{attribute 'linkalways'} 
{attribute 'no_explicit_call' := 'This FB is a CLASS and must be accessed using methods or properties'}
{attribute 'enable_dynamic_creation'}
FUNCTION_BLOCK _ETcVnContourApproximationMethod EXTENDS EnumDatatypeBase
VAR
	localData : ETcVnContourApproximationMethod;
	activeData : REFERENCE TO ETcVnContourApproximationMethod;
	enumBaseDatatype : _DINT(localData);
END_VAR

METHOD PRIVATE AddLocalEnumeration
VAR_INPUT
	Enumeration : T_MAXSTRING;
	Value : ETcVnContourApproximationMethod;
END_VAR
AddEnumeration(Enumeration, Value);
END_METHOD

PROPERTY PUBLIC Address : PVOID
GET
Address := ADR(activeData);
END_GET
END_PROPERTY

METHOD PUBLIC ClearReference
VAR_INPUT
END_VAR
activeData REF= localData;
SetBaseDatatypeReference();
END_METHOD

METHOD PUBLIC Clone : I_Datatype
VAR
    pClone : POINTER TO _ETcVnContourApproximationMethod;
END_VAR
pClone := __NEW(_ETcVnContourApproximationMethod(InitialValue := Value));
Clone := pClone^;
END_METHOD

METHOD FB_init : BOOL
VAR_INPUT
	bInitRetains : BOOL; // if TRUE, the retain variables are initialized (warm start / cold start)
	bInCopyCode : BOOL;  // if TRUE, the instance afterwards gets moved into the copy code (online change)
	InitialValue : ETcVnContourApproximationMethod;
END_VAR
localData := InitialValue;
AddBaseDatatype(enumBaseDatatype);
ClearReference();

AddLocalEnumeration('TCVN_CAM_NONE', ETcVnContourApproximationMethod.TCVN_CAM_NONE);
AddLocalEnumeration('TCVN_CAM_SIMPLE', ETcVnContourApproximationMethod.TCVN_CAM_SIMPLE);
AddLocalEnumeration('TCVN_CAM_TC89_L1', ETcVnContourApproximationMethod.TCVN_CAM_TC89_L1);
AddLocalEnumeration('TCVN_CAM_TC89_KCOS', ETcVnContourApproximationMethod.TCVN_CAM_TC89_KCOS);
END_METHOD

PROPERTY PUBLIC Identifier : T_MAXSTRING
GET
Identifier := 'ETcVnContourApproximationMethod';
END_GET
END_PROPERTY

METHOD IsEnumeratorValueEqual : BOOL
VAR_INPUT
	Enumerator : I_KeyValueForwardEnumerator;
END_VAR
VAR
	storedValue : ETcVnContourApproximationMethod;
END_VAR
IF NOT Enumerator.TryGet(storedValue) THEN
	RETURN;
END_IF

IsEnumeratorValueEqual := storedValue = activeData;
END_METHOD

METHOD PUBLIC MakeReferenceTo
VAR_INPUT
	ReferenceTarget : REFERENCE TO ETcVnContourApproximationMethod;
END_VAR
activeData REF= ReferenceTarget;
SetBaseDatatypeReference();
END_METHOD

METHOD PROTECTED SetBaseDatatypeReference
VAR_INPUT
END_VAR
enumBaseDatatype.MakeReferenceTo(activeData);
END_METHOD

PROPERTY PUBLIC Size : UDINT
GET
Size := SIZEOF(activeData);
END_GET
END_PROPERTY

METHOD TryMakeReferenceTo : BOOL
VAR_INPUT
	Target : I_Datatype;
END_VAR
VAR
	targetAsEnum : I_EnumDatatype;
	pTargetData : POINTER TO ETcVnContourApproximationMethod;
END_VAR
IF NOT Target.TryResolveAsEnumDatatype(targetAsEnum) THEN
	RETURN;
END_IF

IF targetAsEnum.Identifier <> Identifier THEN
	RETURN;
END_IF

pTargetData := Target.Address;
activeData REF= pTargetData^;
SetBaseDatatypeReference();
TryMakeReferenceTo := TRUE;
END_METHOD

PROPERTY PUBLIC Value : ETcVnContourApproximationMethod
GET
Value := activeData;
END_GET
SET
activeData := Value;
END_SET
END_PROPERTY

END_FUNCTION_BLOCK

(* stored: Version 1.1.0.1, ProductVersion 3.1.4024.12
   POU _ETcVnContourApproximationMethod: Id {003f1956-124c-06b3-0455-b539720cc322}, SpecialFunc None
   Folder Constructor: Id {e5ca9629-64ed-0f9e-0668-fc9581229115}
   Folder Private: Id {617f89da-8803-0657-3617-8ccbc4fa3e1e}
   Folder Protected: Id {de9849de-a118-0d95-16f6-4457c88ea99e}
   Method AddLocalEnumeration: Id {45347dc2-f3a3-0e4f-3c10-d473c5cf958f}
   Property Address: Id {23a3061c-bd76-01d4-2c9c-14e8bbea9db4}
   Get Get: Id {154f578b-fcf9-0926-1880-f3799f829073}
   Method ClearReference: Id {b50fb5f7-deb4-0959-0211-9134f834548f}
   Method Clone: Id {e750a80a-b2ed-050c-24f2-d26d747cd782}
   Method FB_init: Id {6a9efe9e-c465-0bcf-01ab-e360e988117c}
   Property Identifier: Id {0d46a558-9bb0-0cd6-3f30-329830ed2e31}
   Get Get: Id {8ee25fef-a62e-0130-0089-b82867ff63c7}
   Method IsEnumeratorValueEqual: Id {e8f24208-2ac0-03de-0164-a2ef46a20e9b}
   Method MakeReferenceTo: Id {dd93ee51-de40-0cc0-0b54-14c113ba02d0}
   Method SetBaseDatatypeReference: Id {5e42cd22-bd84-06fe-09bb-ab0b8f68c82f}
   Property Size: Id {4bd2342e-033c-0fcb-380a-89f2ff2963e0}
   Get Get: Id {36bf6604-d4a0-0eeb-2fc6-8274029d4ec8}
   Method TryMakeReferenceTo: Id {60550a51-7dd8-0ee7-3312-ffb040dd4136}
   Property Value: Id {f8525c58-67bc-023b-076f-1717fd2081f1}
   Get Get: Id {fe9df35c-470f-0cc7-256c-66288330aca9}
   Set Set: Id {4688e632-5726-0c1a-38da-a6a2f19b0251} *)
